// TIA Portal V16 export
// export: Created 2024-03-27T10:00:42.1167192Z, ExportSetting WithDefaults, DisplayName Totally Integrated Automation Portal, DisplayVersion V16, DisplayName TIA Portal Version Control Interface, DisplayVersion V16, DisplayName TIA Portal Openness, DisplayVersion V16, DisplayName STEP 7 Professional, DisplayVersion V16, DisplayName STEP 7 Safety, DisplayVersion V16, DisplayName WinCC Advanced, DisplayVersion V16
TYPE "UR_O2T"
// stored: IsFailsafeCompliant false
   STRUCT
      "Robot IO" { S7_SetPoint := 'True'} : "UR_8_O2T_Robot_IO";
      "Reg 1" { S7_SetPoint := 'True'} : "UR_9_O2T_Registers";
      "Reg 2" { S7_SetPoint := 'True'} : "UR_9_O2T_Registers";
   END_STRUCT;
END_TYPE
